(* CODESYS project M251 Modbus Slave v0.project
   Title: M221 Modbus Slave
   Version: 0.0.0.0
   Author: francisco.florensa

Project tree, tasks and I/O mapping:
  MyController : TM251MESE, Schneider Electric, order no. TM251MESE, version 4.0.6.18
    application Application
      task MAST (cyclic, interval 20 ms, priority 15, watchdog 100 ms x 1) calls MyPOU
      global variables GVL
      program MyPOU [LD]
    IO_Bus : IO bus - TM3, Schneider Electric, version 4.0.6.18
      Module_1 : TM3DI16/G, Schneider Electric, order no. TM3DI16/G, version 1.0.1.4
          input  iwModule_1_IW0 : WORD  // IW0
    COM_Bus : COM bus, Schneider Electric, version 4.0.6.18
    Ethernet_1 : Ethernet Network, Schneider Electric, version 4.0.6.18
        settings: IPAddress = [192, 168, 1, 50]; SubnetMask = [255, 255, 255, 0]; WebServer = TRUE; FTP Server = TRUE; SoMachine Protocol = TRUE; Modbus Server = TRUE; NetManage Protocol = TRUE; SNMP protocol = TRUE; Enable Routing = TRUE; WebVisu protocol = TRUE
    Ethernet_2 : Device Network, Schneider Electric, version 4.0.6.18
        settings: WebServer = TRUE; FTP Server = TRUE; SoMachine Protocol = TRUE; Modbus Server = TRUE; NetManage Protocol = TRUE; SNMP protocol = TRUE; Enable Routing = FALSE; WebVisu protocol = TRUE; DHCP Server Active = TRUE
    Serial_Line_1 : Serial line, Schneider Electric, version 4.0.6.18
      Modbus_Manager : Modbus Manager, Schneider Electric, version 4.0.0.2
*)

// MyController/Application/GVL
VAR_GLOBAL
	data1: INT;
END_VAR
VAR_GLOBAL
	data0 AT %MW0: INT;
END_VAR

// MyController/Application/MyPOU
PROGRAM MyPOU
VAR
END_VAR

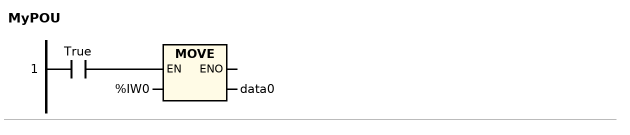
// NETWORK 1
//   data0: AT %MW0
IF True THEN data0 := %IW0; END_IF

END_PROGRAM
